FUNCTION_BLOCK FB_HwRefIOExpander EXTENDS FB_CanNodeBase
VAR_INPUT
END_VAR
VAR_OUTPUT
END_VAR
VAR
	//PDOs
	aInput			AT %I* : ARRAY[1..6] OF UINT;
	aOutput			AT %Q* : ARRAY[1..6] OF UINT;
	
	//Parameter für PulseTrain-Ausgänge
	//aPeriod 		AT %Q* : ARRAY[4..6] OF UINT;
	//aPulse 			AT %Q* : ARRAY[4..6] OF UINT;
	//aPulseNumber 	AT %Q* : ARRAY[4..6] OF UINT;
	aPulseTrainChannel : ARRAY[1..3] OF ST_PulseTrainChannel;

		
END_VAR

IF bNodeEnabled THEN
	SUPER^();
END_IF

ACTION A_ResetApp:
IF nStateA_ResetApp = 0 THEN
	fbSdoWrite(sADSNetID:= stAdsAdress.sNetId, nPortNr:= stAdsAdress.nPort,
				nIndex := cUpdateRequest.nIndex, nSubIndex := 0, nDataLength := 1, nData:= 1, bExecute:= TRUE);
	IF NOT fbSdoWrite.bBusy THEN
		IF fbSdoWrite.bError THEN
			nErrorId := fbSdoWrite.nAdsErrorId;
			nErrorId2 := fbSdoWrite.nSdoErrorId;
			nStateA_ResetApp := 99;  //Error
		ELSE
			nStateA_ResetApp := 80;
		END_IF
		fbSdoWrite(bExecute:= FALSE);
	END_IF
END_IF
END_ACTION

METHOD M_GetPulseTrainChannel : POINTER TO ST_PulseTrainChannel
VAR_INPUT
	nChannel : USINT;
END_VAR
IF nChannel >= 1 AND nChannel <= 3 THEN
	M_GetPulseTrainChannel := ADR(aPulseTrainChannel[nChannel]);
END_IF
END_METHOD

END_FUNCTION_BLOCK

(* stored: Version 1.1.0.1, ProductVersion 3.1.4020.12
   POU FB_HwRefIOExpander: Id {24a32c24-29c4-46dd-a2f6-cf9663d01664}, SpecialFunc None
   Action A_ResetApp: Id {42bc5d37-46f2-49a7-9171-c74c7f582b34}
   Method M_GetPulseTrainChannel: Id {a58362e7-51aa-43e8-9cb3-2846a4e3400f} *)
